// TIA Portal V20 export
FUNCTION "CallSettings" : Void   // FC8, LAD
// Call of settings blocks
// stored: IsIECCheckEnabled true, SetENOAutomatically false
BEGIN

REGION Network 1: Beschreibung / BLOCK INFO HEADER
   // **Betriebsart Automatik / Hand**  
   // Der Baustein ist keiner Betriebsart / Betriebsartenbereich zugeordnet.  
   // 
   // **Alarme**  
   // Der Baustein generiert keine Alarme.  
   // 
   // #### PLC-Datentypen  
   // Verwendete PLC-Datentypen für den SPS-Programmbaustein und das zugehörige WinCC-Bild.  
   // 
   // {.pageWidth}
   // ![Image](CallInterfaceSignals/de/image1.PNG)
   //  
   //  
   // #### Bausteinaufrufe 
   // Der Baustein “LSicar_InterfaceSignalsBool“ wird in diesem FB als Multi-Instanz aufgerufen, entspr. nebenstehender beispielhafter Darstellung.  
   // 
   // {.pageWidth}
   // ![Image](CallInterfaceSignals/de/image2.PNG)
   //  
   // Um einen neuen FB aufzurufen, ziehen Sie den FB in ein neues Netzwerk, wählen Sie „Multiinstanz“ aus, vergeben Sie einen Namen und parametrieren Sie den FB-Aufruf.  
   // 
   // {.pageWidth}
   // ![Image](CallInterfaceSignals/de/image3.PNG)
   //  
   //  
   // #### Weitere Hinweise 
   // 
   // #### Updateinfo 
   // 
   // #### Weitere Dokumente 
   // 
   // ![Icon](_Icon/reference.PNG)
   // 
   // ..\Library Types\LSicar_InterfaceSignalsBool.pdf
   // SIEMENS AG / (c)Copyright 2023
   // ------------------------------------------------------------------------------
   // Title:            CallSettings
   // Comment/Function: Call of SICAR Settings blocks
   // Library/Family:   -
   // Author:           -
   // Tested with:      ---
   // Engineering:      TIA Portal V19
   // Restrictions:     -
   // Requirements:     ---
   // ------------------------------------------------------------------------------
   // Change log table:
   // Version | Date | Expert in charge | Changes applied
   // -------|---------|-------------|--------------------------------------------
   // 01.00.00 | 01.01.1999 | Person x | First released version
   // 01.00.01 | 02.01.1999 | Person y | Block was Updated
END_REGION

REGION Network 2: Set set PLC date and time
   // Change local date and time of the PLC
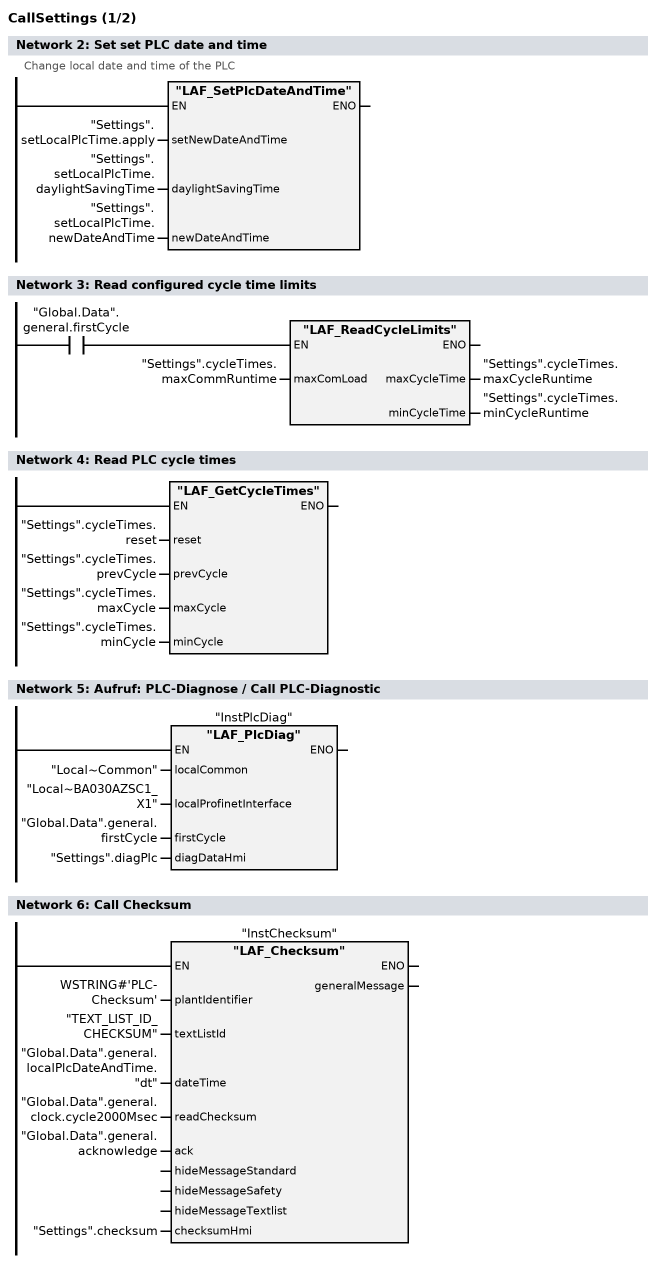
   RUNG wire#powerrail
      "LAF_SetPlcDateAndTime"(setNewDateAndTime := "Settings".setLocalPlcTime.apply, daylightSavingTime := "Settings".setLocalPlcTime.daylightSavingTime, newDateAndTime := "Settings".setLocalPlcTime.newDateAndTime)
   END_RUNG
   // the same network as SCL:
   "LAF_SetPlcDateAndTime"(setNewDateAndTime := "Settings".setLocalPlcTime.apply,
                           daylightSavingTime := "Settings".setLocalPlcTime.daylightSavingTime,
                           newDateAndTime := "Settings".setLocalPlcTime.newDateAndTime);
END_REGION

REGION Network 3: Read configured cycle time limits
   RUNG wire#powerrail
      Contact( "Global.Data".general.firstCycle )
      "LAF_ReadCycleLimits"(maxComLoad := "Settings".cycleTimes.maxCommRuntime, maxCycleTime => "Settings".cycleTimes.maxCycleRuntime, minCycleTime => "Settings".cycleTimes.minCycleRuntime)
   END_RUNG
   // the same network as SCL:
   IF "Global.Data".general.firstCycle THEN
       "LAF_ReadCycleLimits"(maxComLoad := "Settings".cycleTimes.maxCommRuntime,
                             maxCycleTime => "Settings".cycleTimes.maxCycleRuntime,
                             minCycleTime => "Settings".cycleTimes.minCycleRuntime);
   END_IF;
END_REGION

REGION Network 4: Read PLC cycle times
   RUNG wire#powerrail
      "LAF_GetCycleTimes"(reset := "Settings".cycleTimes.reset, prevCycle := "Settings".cycleTimes.prevCycle, maxCycle := "Settings".cycleTimes.maxCycle, minCycle := "Settings".cycleTimes.minCycle)
   END_RUNG
   // the same network as SCL:
   "LAF_GetCycleTimes"(reset := "Settings".cycleTimes.reset,
                       prevCycle := "Settings".cycleTimes.prevCycle,
                       maxCycle := "Settings".cycleTimes.maxCycle,
                       minCycle := "Settings".cycleTimes.minCycle);
END_REGION

REGION Network 5: Aufruf: PLC-Diagnose / Call PLC-Diagnostic
   RUNG wire#powerrail
      "InstPlcDiag"(localCommon := "Local~Common", localProfinetInterface := "Local~BA030AZSC1_X1", firstCycle := "Global.Data".general.firstCycle, diagDataHmi := "Settings".diagPlc)
   END_RUNG
   // the same network as SCL:
   "InstPlcDiag"(localCommon := "Local~Common",   // "LAF_PlcDiag"
                 localProfinetInterface := "Local~BA030AZSC1_X1",
                 firstCycle := "Global.Data".general.firstCycle,
                 diagDataHmi := "Settings".diagPlc);
END_REGION

REGION Network 6: Call Checksum
   RUNG wire#powerrail
      "InstChecksum"(plantIdentifier := WSTRING#'PLC-Checksum', textListId := "TEXT_LIST_ID_CHECKSUM", dateTime := "Global.Data".general.localPlcDateAndTime."dt", readChecksum := "Global.Data".general.clock.cycle2000Msec, ack := "Global.Data".general.acknowledge, hideMessageStandard :=, hideMessageSafety :=, hideMessageTextlist :=, checksumHmi := "Settings".checksum, generalMessage =>)
   END_RUNG
   // the same network as SCL:
   "InstChecksum"(plantIdentifier := WSTRING#'PLC-Checksum',   // "LAF_Checksum"
                  textListId := "TEXT_LIST_ID_CHECKSUM",
                  dateTime := "Global.Data".general.localPlcDateAndTime."dt",
                  readChecksum := "Global.Data".general.clock.cycle2000Msec,
                  ack := "Global.Data".general.acknowledge,
                  checksumHmi := "Settings".checksum);
END_REGION

REGION Network 7: Aufruf: SMC-Diagnose (SIMATIC Memory Card - Diagnose) / Call SMC-Diagnostic (SIMATIC Memory Card - Diagnostic)
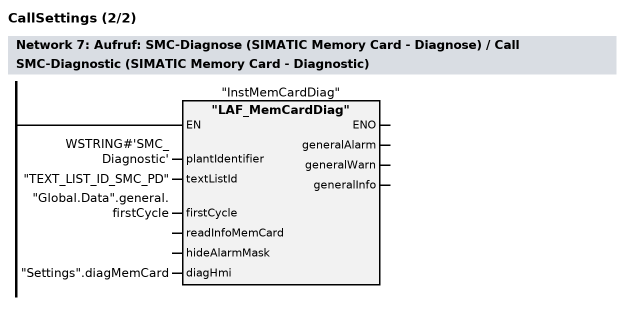
   RUNG wire#powerrail
      "InstMemCardDiag"(plantIdentifier := WSTRING#'SMC_Diagnostic', textListId := "TEXT_LIST_ID_SMC_PD", firstCycle := "Global.Data".general.firstCycle, readInfoMemCard :=, hideAlarmMask :=, diagHmi := "Settings".diagMemCard, generalAlarm =>, generalWarn =>, generalInfo =>)
   END_RUNG
   // the same network as SCL:
   "InstMemCardDiag"(plantIdentifier := WSTRING#'SMC_Diagnostic',   // "LAF_MemCardDiag"
                     textListId := "TEXT_LIST_ID_SMC_PD",
                     firstCycle := "Global.Data".general.firstCycle,
                     diagHmi := "Settings".diagMemCard);
END_REGION
END_FUNCTION
